VISUALIZATION about  // 800x480
END_VISUALIZATION

(* stored: Version 1.1.0.1, ProductVersion 3.1.4018.5
   Visu about: Id {a1fd3a7a-3e01-4be3-ab09-73779677c149} *)
